(* IEC 61131-3 sources: BRUSdevice/, 4 files *)

(* ---- Types.typ ---- *)
TYPE
	CIFSDevChkInfo_typ : 	STRUCT
		Status : STRING[80]; (*Detail string for status of function block*)
		StatusID : CIFSDevChkStatusID_enum;
		State : CIFSDevChk_enum; (*Internal operating step of the function block*)
		fileIOStatus : UINT;
	END_STRUCT;
	CIFSDevChkPar_typ : 	STRUCT
		DeviceName : STRING[80]; (*Optional device name. If left blank, the name of the created USB device will be 'USBDEV1'*)
		ServerDomain : STRING[80];
		ServerPw : STRING[80];
		ServerUser : STRING[80];
		ServerIP : STRING[80];
		ShareName : STRING[80];
	END_STRUCT;
	CIFSDevChkStatusID_enum :
		(
		cifsdevERR_OK := 0, (*No errors*)
		cifsdevERR_AUTOLINK_PARAM := 10000,
		cifsdevERR_NO_USB_FOUND := 10001 (*Shown if a link was attempted, but no mass storage devices were found.*)
		);
	CIFSDevChk_enum :
		(
		CIFS_IDLE,
		CIFS_LINK,
		CIFS_LINKED,
		CIFS_UNLINK,
		CIFS_ERROR
		);
	USBDevChkInfo_typ : 	STRUCT
		Status : STRING[80]; (*Detail string for status of function block*)
		StatusID : USBDevChkStatusID_enum;
		State : USBDevChk_enum; (*Internal operating step of the function block*)
		DiskSizeBytes : UDINT; (*Total memory size of connected device in bytes*)
		FreeMemBytes : UDINT; (*Amount of memory available in bytes*)
	END_STRUCT;
	USBDevChkPar_typ : 	STRUCT
		AutoLink : BOOL; (*When set high, function will try to link to a mass storage device at a set interval*)
		AutoLinkInterval : TIME; (*When autolink is enabled, how long between checks for devices*)
		DeviceName : STRING[80]; (*Optional device name. If left blank, the name of the created USB device will be 'USBDEV1'*)
	END_STRUCT;
	USBDevChkStatusID_enum :
		(
		usbdevERR_OK := 0, (*No errors*)
		usbdevERR_AUTOLINK_PARAM := 10000,
		usbdevERR_NO_USB_FOUND := 10001 (*Shown if a link was attempted, but no mass storage devices were found.*)
		);
	USBDevChk_enum :
		(
		USB_IDLE,
		USB_NODE_LIST,
		USB_NODE_GET,
		USB_LINK,
		USB_MEMINFO,
		USB_LINKED,
		USB_UNLINK,
		USB_ERROR
		);
	zzCIFSInternalStruct_typ : 	STRUCT  (* *) (* *) (*#OMIT*)
		step : CIFSDevChk_enum;
		cmd : zzCIFS_cmd_typ;
		par : zzCIFS_par_typ;
		stat : zzCIFS_stat_typ;
		fb : zzCIFS_fb_typ;
		old : zzCIFS_old;
	END_STRUCT;
	zzCIFS_cmd_typ : 	STRUCT  (* *) (* *) (*#OMIT*)
		link : BOOL;
	END_STRUCT;
	zzCIFS_fb_typ : 	STRUCT  (* *) (* *) (*#OMIT*)
		devLink : DevLink;
		devUnlink : DevUnlink;
		errorReset : TON;
		linkTimeout : TON;
	END_STRUCT;
	zzCIFS_old : 	STRUCT  (* *) (* *) (*#OMIT*)
		enable : BOOL;
		link : BOOL;
		eject : BOOL;
		update : BOOL;
	END_STRUCT;
	zzCIFS_par_typ : 	STRUCT  (* *) (* *) (*#OMIT*)
		devName : STRING[80] := 'USBDEV1';
		parStrFull : STRING[150] := '/DEVICE=';
		handle : UDINT;
		emptyStr : STRING[80] := '';
		user : CIFSDevChkPar_typ;
	END_STRUCT;
	zzCIFS_stat_typ : 	STRUCT  (* *) (* *) (*#OMIT*)
		ready : BOOL;
		initDone : BOOL;
	END_STRUCT;
	zzUSBInternalStruct_typ : 	STRUCT  (* *) (* *) (*#OMIT*)
		step : USBDevChk_enum;
		cmd : zzUSB_cmd_typ;
		par : zzUSB_par_typ;
		stat : zzUSB_stat_typ;
		fb : zzUSB_fb_typ;
		old : zzUSB_old;
	END_STRUCT;
	zzUSB_cmd_typ : 	STRUCT  (* *) (* *) (*#OMIT*)
		link : BOOL;
		autoLink : BOOL;
	END_STRUCT;
	zzUSB_fb_typ : 	STRUCT  (* *) (* *) (*#OMIT*)
		devLink : DevLink;
		devUnlink : DevUnlink;
		UsbNodeListGet : UsbNodeListGet;
		UsbNodeGet : UsbNodeGet;
		autoLink : TON;
		errorReset : TON;
		nodeSearchTimeout : TON;
		DevMemInfo : DevMemInfo;
	END_STRUCT;
	zzUSB_old : 	STRUCT  (* *) (* *) (*#OMIT*)
		enable : BOOL;
		link : BOOL;
		eject : BOOL;
		update : BOOL;
	END_STRUCT;
	zzUSB_par_typ : 	STRUCT  (* *) (* *) (*#OMIT*)
		devName : STRING[80] := 'USBDEV1';
		parStrFull : STRING[150] := '/DEVICE=';
		nodeList : ARRAY[0..3]OF UDINT;
		nodeInfo : usbNode_typ;
		handle : UDINT;
		emptyStr : STRING[80] := '';
		user : USBDevChkPar_typ;
		node : USINT;
	END_STRUCT;
	zzUSB_stat_typ : 	STRUCT  (* *) (* *) (*#OMIT*)
		ready : BOOL;
		initDone : BOOL;
	END_STRUCT;
END_TYPE

(* ---- CIFSDevChk.st ---- *)
(* Links to CIFS devices at runtime and creates a file device. *)
FUNCTION_BLOCK CIFSDevChk

	// Initialization routine
	IF Enable AND NOT(IS.stat.initDone) THEN
		// check parameters
		IF FALSE THEN
			(*possible parameter checking*)
		ELSE
			// make par string
			IS.par.parStrFull := '/SIP=';
			brsstrcat(ADR(IS.par.parStrFull), ADR(Parameters.ServerIP));

			brsstrcat(ADR(IS.par.parStrFull), ADR(' /PROTOCOL=cifs'));

			IF brsstrcmp(ADR(Parameters.ServerDomain), ADR('')) = 0 THEN
				// Do not add the domain tag
			ELSE
				brsstrcat(ADR(IS.par.parStrFull), ADR(' /DOMAIN='));
				brsstrcat(ADR(IS.par.parStrFull), ADR(Parameters.ServerDomain));
			END_IF

			brsstrcat(ADR(IS.par.parStrFull), ADR(' /SHARE='));
			brsstrcat(ADR(IS.par.parStrFull), ADR(Parameters.ShareName));

			brsstrcat(ADR(IS.par.parStrFull), ADR(' /USER='));
			brsstrcat(ADR(IS.par.parStrFull), ADR(Parameters.ServerUser));

			brsstrcat(ADR(IS.par.parStrFull), ADR(' /PASSWORD='));
			brsstrcat(ADR(IS.par.parStrFull), ADR(Parameters.ServerPw));

			// load in device pars
			IF brsstrcmp(ADR(Parameters.DeviceName), ADR(IS.par.emptyStr)) = 0 THEN
				IS.par.devName	:= 'CIFSDEV1';
			ELSE
				IS.par.devName	:= Parameters.DeviceName;
			END_IF

			// go to run mode
			IS.stat.initDone	:= TRUE;
			Info.Status			:= 'Init OK';
			Info.StatusID		:= cifsdevERR_OK;
		END_IF
	// Cyclic operation
	ELSIF IS.stat.initDone THEN

		// read in commands (edge sensitive)
		IS.cmd.link := Link AND NOT(IS.old.link);

		// state machine
		CASE IS.step OF
			CIFS_IDLE:
				IF IS.cmd.link THEN
					IS.step				:= CIFS_LINK;
					Info.StatusID		:= cifsdevERR_OK;
					Info.StatusID		:= 0;
					IS.cmd.link			:= FALSE;
				ELSIF (Eject OR NOT(Enable)) AND Ready THEN
					Info.Status			:= 'Disconnecting...';
					IS.step				:= CIFS_UNLINK;
				ELSIF NOT Enable OR (Update AND NOT IS.old.update) THEN
					IS.stat.initDone	:= FALSE;
				END_IF

			CIFS_LINK:
				IS.fb.devLink.pParam	:= ADR(IS.par.parStrFull); // string of device pars (see help)
				IS.fb.devLink.pDevice	:= ADR(IS.par.devName); // name of the created device
				IS.fb.devLink.enable	:= TRUE;

				IF IS.fb.devLink.status = ERR_FUB_BUSY OR IS.fb.devLink.status = ERR_FUB_ENABLE_FALSE THEN
					// do nothing, stay in state
				ELSIF IS.fb.devLink.status = ERR_OK THEN
					// success, move to grab mem info
					IS.step					:= CIFS_LINKED;
					IS.par.handle			:= IS.fb.devLink.handle;
					IS.fb.devLink.enable	:= FALSE;
					Info.Status				:= 'CIFS Share Connected';

				ELSE
					Info.fileIOStatus		:= FileIoGetSysError();
					Info.Status				:= 'ERR: Error connecting to device!';
					IS.step					:= CIFS_ERROR;
					IS.fb.devLink.enable	:= FALSE;
				END_IF

			CIFS_LINKED:
				// wait to be unlinked
				IF Eject OR (NOT Enable) THEN
					IS.step	:= CIFS_UNLINK;
				END_IF

			CIFS_UNLINK:
				IS.fb.devUnlink.handle	:= IS.par.handle;
				IS.fb.devUnlink.enable	:= TRUE;

				IF IS.fb.devUnlink.status = ERR_FUB_BUSY OR IS.fb.devUnlink.status = ERR_FUB_ENABLE_FALSE THEN
					// do nothing, stay in state
				ELSIF IS.fb.devUnlink.status = ERR_OK THEN
					// success, move on
					IS.step				:= CIFS_IDLE;
					Info.Status			:= 'Disconnected';

					IS.fb.devUnlink.enable	:= FALSE;

					// de-init the function block if disabled
					IF NOT Enable THEN
						IS.stat.initDone	:= FALSE;
					END_IF
				ELSE
					Info.Status				:= 'ERR: Error in disconnecting!';
					IS.step					:= CIFS_ERROR;
					IS.fb.devUnlink.enable	:= FALSE;
				END_IF

			CIFS_ERROR:
				IF ErrorReset THEN
					IS.fb.devLink.enable		:= FALSE;
					IS.fb.devUnlink.enable		:= FALSE;
					IS.step						:= CIFS_IDLE;
					Info.Status					:= 'Reset OK';
					Info.StatusID				:= cifsdevERR_OK;
				ELSIF NOT Enable THEN
					IS.stat.initDone			:= FALSE;
				END_IF

		END_CASE;

		// call device related functions
		IS.fb.devLink();
		IS.fb.devUnlink();

		// reject update commands
		IF Update AND NOT IS.old.update AND IS.step <> CIFS_IDLE THEN
			Info.Status			:= 'Update failed - State must be Idle';
		END_IF

	END_IF

	// FUNCTION BLOCK DISABLED AND EJECTED
	IF NOT(Enable) AND NOT(IS.stat.initDone) THEN
		IS.step				:= CIFS_IDLE;
		Info.State			:= IS.step;
		Error				:= FALSE;
		Info.StatusID		:= cifsdevERR_OK;
		Info.Status			:= 'Function block disabled';
	END_IF

	// set edge detection variables
	IS.old.eject	:= Eject;
	IS.old.link		:= Link;
	IS.old.enable	:= Enable;
	IS.old.update	:= Update;

	// set function outputs
	Info.State		:= IS.step;
	Active			:= IS.stat.initDone;
	Error			:= IS.step = CIFS_ERROR;
	Ready			:= IS.step = CIFS_LINKED;

END_FUNCTION_BLOCK

(* ---- USBDevChk.st ---- *)
(* Checks for and links to USB devices at runtime and creates a file device. *)
FUNCTION_BLOCK USBDevChk

	// Initialization routine
	IF Enable AND NOT(IS.stat.initDone) THEN
		// check parameters
		IF Parameters.AutoLink AND Parameters.AutoLinkInterval < T#2s THEN
			Info.Status	:= 'WARN: AutoLinkInvterval must be >2s';
			Info.StatusID	:= usbdevERR_AUTOLINK_PARAM;
		ELSE
			// load in device pars
			IF brsstrcmp(ADR(Parameters.DeviceName), ADR(IS.par.emptyStr)) = 0 THEN
				IS.par.devName	:= 'USBDEV1';
			ELSE
				IS.par.devName	:= Parameters.DeviceName;
			END_IF
			IS.par.user.AutoLinkInterval	:= Parameters.AutoLinkInterval;
			IS.par.user.AutoLink			:= Parameters.AutoLink;
			// go to run mode
			IS.stat.initDone	:= TRUE;
			Info.Status			:= 'Init OK';
			Info.StatusID		:= usbdevERR_OK;
			IS.par.node			:= 0;
		END_IF
	// Cyclic operation
	ELSIF IS.stat.initDone THEN

		// read in commands (edge sensitive)
		IS.cmd.link		:= Link AND NOT IS.old.link;
		IS.cmd.autoLink	:= IS.fb.autoLink.Q;

		// state machine
		CASE IS.step OF
			USB_IDLE:
				IF IS.cmd.link OR IS.cmd.autoLink THEN
					IS.step				:= USB_NODE_LIST;
					Info.StatusID		:= usbdevERR_OK;
					IS.par.node			:= 0;
					Info.StatusID		:= 0;
					IS.cmd.link			:= FALSE;
					IS.cmd.autoLink		:= FALSE;
				ELSIF (Eject OR NOT(Enable)) AND Ready THEN
					Info.Status			:= 'USB Ejecting...';
					IS.step				:= USB_UNLINK;
				ELSIF NOT Enable THEN
					IS.stat.initDone	:= FALSE;
				END_IF

			USB_NODE_LIST:
				IS.fb.UsbNodeListGet.enable						:= TRUE;
				IS.fb.UsbNodeListGet.bufferSize					:= SIZEOF(IS.par.nodeList);
				IS.fb.UsbNodeListGet.filterInterfaceClass		:= asusb_CLASS_MASS_STORAGE;
				IS.fb.UsbNodeListGet.filterInterfaceSubClass	:= 0;
				IS.fb.UsbNodeListGet.pBuffer					:= ADR(IS.par.nodeList);

				IF IS.fb.UsbNodeListGet.listNodes > 0 AND IS.fb.UsbNodeListGet.status = ERR_OK THEN
					IS.step						:= USB_NODE_GET;
					IS.fb.UsbNodeListGet.enable	:= FALSE;
				ELSIF IS.fb.nodeSearchTimeout.Q OR IS.fb.UsbNodeListGet.status = asusbERR_USB_NOTFOUND THEN
					IS.step						:= USB_IDLE;
					IS.fb.UsbNodeListGet.enable	:= FALSE;
					Info.Status					:= 'WARN: No USB device found!';
					Info.StatusID				:= usbdevERR_NO_USB_FOUND;
				ELSIF IS.fb.UsbNodeListGet.status = ERR_FUB_ENABLE_FALSE OR IS.fb.UsbNodeListGet.status = ERR_FUB_BUSY THEN
					// do nothing
				ELSE
					IS.step						:= USB_ERROR;
					IS.fb.UsbNodeListGet.enable	:= FALSE;
				END_IF

			USB_NODE_GET:
				IS.fb.UsbNodeGet.enable		:= TRUE;
				IS.fb.UsbNodeGet.bufferSize	:= SIZEOF(IS.par.nodeInfo);
				IS.fb.UsbNodeGet.nodeId		:= IS.par.nodeList[IS.par.node];
				IS.fb.UsbNodeGet.pBuffer	:= ADR(IS.par.nodeInfo);

				IF IS.fb.UsbNodeGet.status = ERR_OK THEN
					IS.step					:= USB_LINK;
					IS.fb.UsbNodeGet.enable	:= FALSE;

					IS.par.parStrFull		:= '/DEVICE=';
					brsstrcat(ADR(IS.par.parStrFull), ADR(IS.par.nodeInfo.ifName));
				ELSIF IS.fb.nodeSearchTimeout.Q OR IS.fb.UsbNodeListGet.status = asusbERR_USB_NOTFOUND THEN
					IS.step					:= USB_IDLE;
					IS.fb.UsbNodeGet.enable	:= FALSE;
					Info.Status				:= 'WARN: No USB device found!';
					Info.StatusID			:= usbdevERR_NO_USB_FOUND;
				ELSIF IS.fb.UsbNodeGet.status = ERR_FUB_ENABLE_FALSE OR IS.fb.UsbNodeGet.status = ERR_FUB_BUSY THEN
					// do nothing
				ELSE
					IS.step					:= USB_ERROR;
					IS.fb.UsbNodeGet.enable	:= FALSE;
				END_IF

			USB_LINK:
				IS.fb.devLink.pParam	:= ADR(IS.par.parStrFull); // string of device pars (see help)
				IS.fb.devLink.pDevice	:= ADR(IS.par.devName); // name of the created device
				IS.fb.devLink.enable	:= TRUE;

				IF IS.fb.devLink.status = ERR_FUB_BUSY OR IS.fb.devLink.status = ERR_FUB_ENABLE_FALSE THEN
					// do nothing, stay in state
				ELSIF IS.fb.devLink.status = ERR_OK THEN
					// success, move to grab mem info
					IS.step					:= USB_MEMINFO;
					IS.par.handle			:= IS.fb.devLink.handle;
					IS.fb.devLink.enable	:= FALSE;
					Info.Status				:= 'USB Device Linked';
				ELSE
					Info.Status				:= 'ERR: Error connecting to device!';
					IS.step					:= USB_ERROR;
					IS.fb.devLink.enable	:= FALSE;
				END_IF

			USB_MEMINFO:
				IF IS.fb.DevMemInfo.status = ERR_OK THEN
					IS.step				:= USB_LINKED;
					Info.DiskSizeBytes	:= IS.fb.DevMemInfo.memsize;
					Info.FreeMemBytes	:= IS.fb.DevMemInfo.freemem;

					IF IS.fb.DevMemInfo.freemem = 0 THEN
						IS.par.node	:= IS.par.node + 1;
						IS.step		:= USB_UNLINK;
					END_IF
				ELSIF IS.fb.DevMemInfo.status <> ERR_FUB_BUSY AND IS.fb.DevMemInfo.status <> ERR_FUB_ENABLE_FALSE THEN
					IS.step			:= USB_ERROR;
					Info.Status		:= 'ERR: Error reading device memory information';
				END_IF

			USB_LINKED:
				// wait to be unlinked
				IF Eject OR (NOT Enable) THEN
					IS.step	:= USB_UNLINK;
				END_IF

			USB_UNLINK:
				IS.fb.devUnlink.handle	:= IS.par.handle;
				IS.fb.devUnlink.enable	:= TRUE;

				IF IS.fb.devUnlink.status = ERR_FUB_BUSY OR IS.fb.devUnlink.status = ERR_FUB_ENABLE_FALSE THEN
					// do nothing, stay in state
				ELSIF IS.fb.devUnlink.status = ERR_OK THEN
					// success, move on
					IF NOT Eject AND IS.par.node < usbdevMAX_NODES AND IS.par.nodeList[IS.par.node] <> 0 THEN
						IS.step				:= USB_NODE_GET;
					ELSIF IS.par.node >= usbdevMAX_NODES OR IS.par.nodeList[IS.par.node] = 0 THEN
						IS.step				:= USB_IDLE;
						Info.Status			:= 'No suitable USB detected!';
						Info.StatusID		:= usbdevERR_NO_USB_FOUND;
						IS.par.node			:= 0;
					ELSE
						IS.step				:= USB_IDLE;
						Info.Status			:= 'USB Device Ejected';
					END_IF
					IS.fb.devUnlink.enable	:= FALSE;
					Info.DiskSizeBytes		:= 0;
					Info.FreeMemBytes		:= 0;

					// de-init the function block if disabled
					IF NOT Enable THEN
						IS.stat.initDone	:= FALSE;
					END_IF
				ELSE
					Info.Status				:= 'ERR: Error unlinking device!';
					IS.step					:= USB_ERROR;
					IS.fb.devUnlink.enable	:= FALSE;
				END_IF

			USB_ERROR:
				IF ErrorReset THEN
					IS.fb.devLink.enable		:= FALSE;
					IS.fb.devUnlink.enable		:= FALSE;
					IS.fb.UsbNodeGet.enable		:= FALSE;
					IS.fb.UsbNodeListGet.enable	:= FALSE;
					IS.step						:= USB_IDLE;
					Info.Status					:= 'Reset OK';
					IS.par.node					:= 0;
					Info.StatusID				:= usbdevERR_OK;
				ELSIF NOT Enable THEN
					IS.stat.initDone			:= FALSE;
				END_IF

		END_CASE;

		// call device related functions
		IS.fb.devLink();
		IS.fb.devUnlink();
		IS.fb.UsbNodeGet();
		IS.fb.UsbNodeListGet();

		// call timers
		IS.fb.autoLink(IN := IS.par.user.AutoLink  AND IS.step = USB_IDLE AND NOT(Eject) AND Enable, PT := IS.par.user.AutoLinkInterval);
		IS.fb.nodeSearchTimeout(IN := ((IS.step = USB_NODE_GET OR IS.step = USB_NODE_LIST) AND Enable), PT := T#5s);

		// check for update commands
		IF Update AND NOT IS.old.update THEN
			IS.stat.initDone		:= FALSE;

			// if a device is already connected, the Update command should also update the amount of available memory
			IF IS.step = USB_LINKED THEN
				IS.step	:= USB_MEMINFO;
			END_IF
		END_IF

		// gather information about the device when requested
		IS.fb.DevMemInfo.enable		:= (IS.step = USB_MEMINFO);
		IS.fb.DevMemInfo.pDevice	:= ADR(IS.par.devName);
		IS.fb.DevMemInfo();
	END_IF

	// FUNCTION BLOCK DISABLED AND EJECTED
	IF NOT(Enable) AND NOT(IS.stat.initDone) THEN
		IS.step				:= USB_IDLE;
		Info.State			:= IS.step;
		Error				:= FALSE;
		IS.par.node			:= 0;
		Info.DiskSizeBytes	:= 0;
		Info.FreeMemBytes	:= 0;
		Info.StatusID		:= usbdevERR_OK;
		Info.Status			:= 'Function block disabled';
	END_IF

	// set edge detection variables
	IS.old.eject	:= Eject;
	IS.old.link		:= Link;
	IS.old.enable	:= Enable;
	IS.old.update	:= Update;

	// set function outputs
	Info.State		:= IS.step;
	Active			:= IS.stat.initDone;
	Error			:= IS.step = USB_ERROR;
	Ready			:= IS.step = USB_LINKED;

END_FUNCTION_BLOCK

(* ---- Constants.var ---- *)
VAR CONSTANT
	usbdevMAX_NODES : USINT := 4; (*Maximum number of USB ports that will be checked*)
END_VAR
